TYPE S_Command_Control :
STRUCT
	// Input
	Command AT %Q* : UINT;
	
	// output
	CurrentJobID AT %I* : UINT;
END_STRUCT
END_TYPE

(* stored: Version 1.1.0.1, ProductVersion 3.1.4024.10
   DUT S_Command_Control: Id {7862e245-a319-42a1-bb82-4868c813c623} *)
